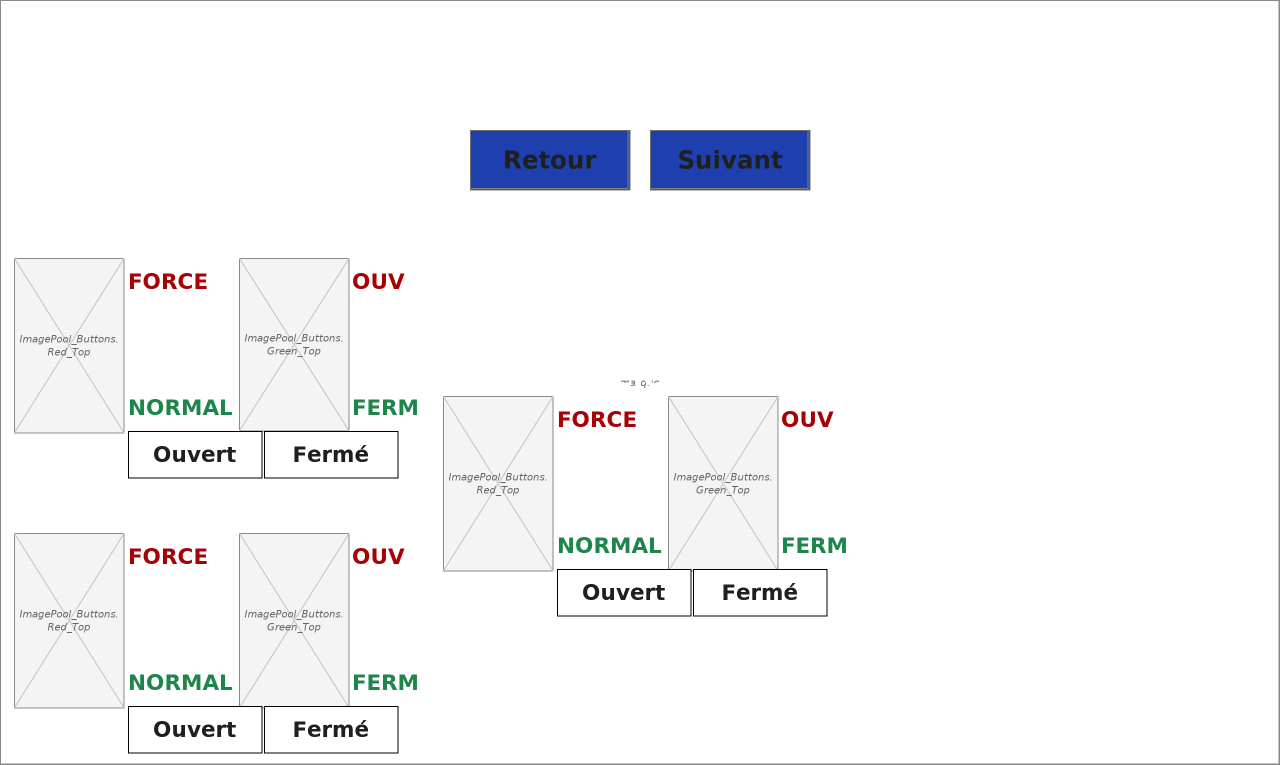
VISUALIZATION Maintenance_4  // 1280x765
    Frame (0,0 1280x765)
        shows masque()
    Button (470,130 160x60), "Retour"
        OnMouseDown: execute {
            IF (Option_Bas_Debit OR Option_Douchette OR Option_NEP)
            	THEN
            	VisuElems.CURRENTVISU := 'Maintenance_3';
            	ELSIF (Option_Douche OR Option_Lavabo)
            		THEN
            		VisuElems.CURRENTVISU := 'Maintenance_2';
            	ELSIF (Option_RegSouf_Ultrason OR Option_Reg_Etanche_Ext OR Option_V3V_EauMitig)
            		THEN
            		VisuElems.CURRENTVISU := 'Maintenance_1';
            	ELSE
            	VisuElems.CURRENTVISU := 'menu';
            END_IF
        }
    Button (650,130 160x60), "Suivant"
        OnMouseDown: execute {
            IF (Option_Cabine_Climatique)
            	THEN
            	VisuElems.CURRENTVISU := 'Maintenance_5';
            	ELSIF (Option_Com_RegSouf_Ultrason)
            		THEN
            		VisuElems.CURRENTVISU := 'Maintenance_6';
            	ELSE
            		VisuElems.CURRENTVISU := 'Maintenance_7';
            END_IF
        }
    Group (14,218 415x260), invisible if: NOT Option_WC_GV
        Group (0,40 415x173)
            Group (0,0 225x173)
                Group (0,0 110x175)
                    Image (0,0 110x175), text variable: EF_Cmd_Verin_WC_GV, invisible if: EF_Cmd_Verin_WC_GV, image: ImagePool_Buttons.Green_Bottom
                        OnMouseDown: toggle EF_Cmd_Verin_WC_GV
                    Image (0,0 110x175), text variable: NOT EF_Cmd_Verin_WC_GV, invisible if: NOT EF_Cmd_Verin_WC_GV, image: ImagePool_Buttons.Red_Top
                        OnMouseDown: toggle EF_Cmd_Verin_WC_GV
                Rectangle (111,0 114x47), "FORCE"
                Rectangle (111,63 114x47), "MODE"
                Rectangle (111,126 114x47), "NORMAL"
            Group (225,0 190x173), invisible if: NOT EF_Cmd_Verin_WC_GV
                Group (0,0 110x173)
                    Image (0,0 110x173), invisible if: F_Cmd_Verin_WC_GV, image: ImagePool_Buttons.Red_Bottom
                        OnMouseDown: toggle F_Cmd_Verin_WC_GV
                    Image (0,0 110x173), invisible if: NOT F_Cmd_Verin_WC_GV, image: ImagePool_Buttons.Green_Top
                        OnMouseDown: toggle F_Cmd_Verin_WC_GV
                Rectangle (110,0 80x47), "OUV"
                Rectangle (110,63 80x47), "OUT"
                Rectangle (110,126 80x47), "FERM"
        Group (34,213 350x47), invisible if: TRUE
            Rectangle (0,0 80x47), "FDC :"
            RoundedRectangle (80,0 134x47), "Ouvert"
            RoundedRectangle (216,0 134x47), "Fermé"
        Rectangle (0,0 415x40), "Chasse WC gros volume"
    Group (14,493 415x260), invisible if: NOT Option_WC_PV
        Group (0,40 415x173)
            Group (0,0 225x173)
                Group (0,0 110x175)
                    Image (0,0 110x175), invisible if: EF_Cmd_Verin_WC_PV, image: ImagePool_Buttons.Green_Bottom
                        OnMouseDown: toggle EF_Cmd_Verin_WC_PV
                    Image (0,0 110x175), invisible if: NOT EF_Cmd_Verin_WC_PV, image: ImagePool_Buttons.Red_Top
                        OnMouseDown: toggle EF_Cmd_Verin_WC_PV
                Rectangle (111,0 114x47), "FORCE"
                Rectangle (111,63 114x47), "MODE"
                Rectangle (111,126 114x47), "NORMAL"
            Group (225,0 190x173), invisible if: NOT EF_Cmd_Verin_WC_PV
                Group (0,0 110x175)
                    Image (0,0 110x175), invisible if: F_Cmd_Verin_WC_PV, image: ImagePool_Buttons.Red_Bottom
                        OnMouseDown: toggle F_Cmd_Verin_WC_PV
                    Image (0,0 110x175), invisible if: NOT F_Cmd_Verin_WC_PV, image: ImagePool_Buttons.Green_Top
                        OnMouseDown: toggle F_Cmd_Verin_WC_PV
                Rectangle (110,0 80x47), "OUV"
                Rectangle (110,63 80x47), "OUT"
                Rectangle (110,126 80x47), "FERM"
        Group (34,213 350x47), invisible if: TRUE
            Rectangle (0,0 80x47), "FDC :"
            RoundedRectangle (80,0 134x47), "Ouvert"
            RoundedRectangle (216,0 134x47), "Fermé"
        Rectangle (0,0 415x40), "Chasse WC petit volume"
    Group (443,356 415x260), invisible if: NOT Option_Prise
        Group (0,40 415x173)
            Group (0,0 225x173)
                Group (0,0 110x175)
                    Image (0,0 110x175), invisible if: EF_Cmd_PC_Cab, image: ImagePool_Buttons.Green_Bottom
                        OnMouseDown: toggle EF_Cmd_PC_Cab
                    Image (0,0 110x175), invisible if: NOT EF_Cmd_PC_Cab, image: ImagePool_Buttons.Red_Top
                        OnMouseDown: toggle EF_Cmd_PC_Cab
                Rectangle (111,0 114x47), "FORCE"
                Rectangle (111,63 114x47), "MODE"
                Rectangle (111,126 114x47), "NORMAL"
            Group (225,0 190x173), invisible if: NOT EF_Cmd_PC_Cab
                Group (0,0 110x175)
                    Image (0,0 110x175), invisible if: F_Cmd_PC_Cab, image: ImagePool_Buttons.Red_Bottom
                        OnMouseDown: toggle F_Cmd_PC_Cab
                    Image (0,0 110x175), invisible if: NOT F_Cmd_PC_Cab, image: ImagePool_Buttons.Green_Top
                        OnMouseDown: toggle F_Cmd_PC_Cab
                Rectangle (110,0 80x47), "OUV"
                Rectangle (110,63 80x47), "OUT"
                Rectangle (110,126 80x47), "FERM"
        Group (34,213 350x47), invisible if: TRUE
            Rectangle (0,0 80x47), "FDC :"
            RoundedRectangle (80,0 134x47), "Ouvert"
            RoundedRectangle (216,0 134x47), "Fermé"
        Rectangle (0,0 415x40), "Prise électrique"
END_VISUALIZATION

(* stored: Version 1.1.0.1, ProductVersion 3.1.4024.15
   Visu Maintenance_4: Id {c842a447-ce2c-4581-a851-4e764a52897a} *)
